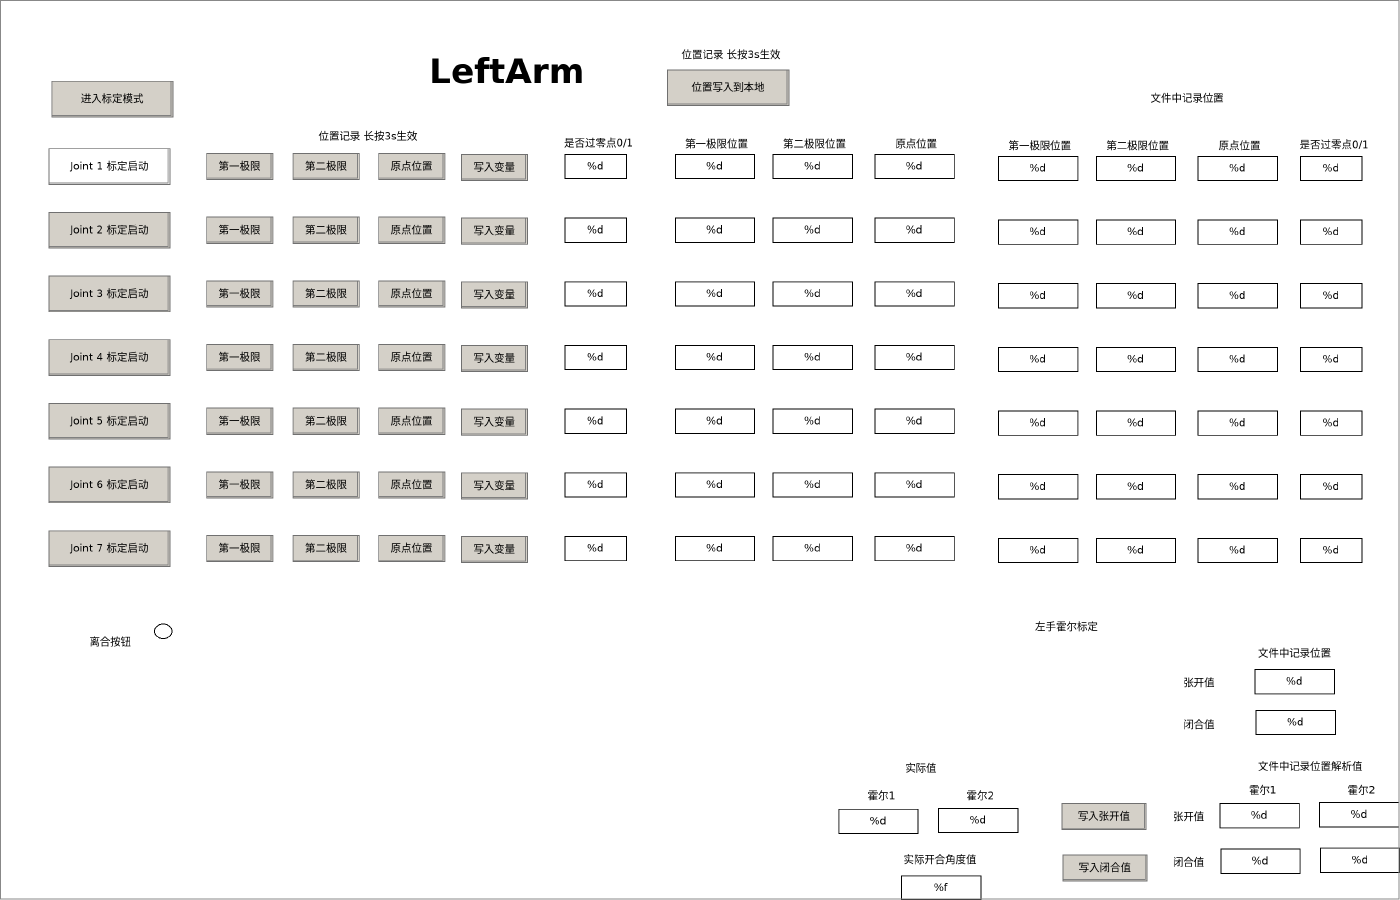
VISUALIZATION LeftArmCali  // 1473x947
    Button (54,85 128x38), "进入标定模式", colour toggle: GVL_armCali.g_armEnterCaliMode[1]
        toggle GVL_armCali.g_armEnterCaliMode[1]
    Button (51,156 128x38), "Joint 1 标定启动", colour toggle: GVL_armCali.g_jointIntoCaliState[1][1]
        toggle GVL_armCali.g_jointIntoCaliState[1][1]
    Label (435,49 197x52), "LeftArm"
    Button (51,223 128x38), "Joint 2 标定启动", colour toggle: GVL_armCali.g_jointIntoCaliState[1][2]
        toggle GVL_armCali.g_jointIntoCaliState[1][2]
    Button (217,161 70x28), "第一极限", colour toggle: GVL_armCali.g_linkEncFristCaliTrigger[1][1]
        tap GVL_armCali.g_linkEncFristPosCali[1][1]
    Button (308,161 70x28), "第二极限", colour toggle: GVL_armCali.g_linkEncSecondCaliTrigger[1][1]
        tap GVL_armCali.g_linkEncSecondPosCali[1][1]
    Rectangle (594,162 65x26), "%d", text variable: GVL_armCali.g_linkZeroCrossOrNot[1][1]
    Label (589,139 82x23), "是否过零点0/1"
    Rectangle (710,162 84x26), "%d", text variable: GVL_armCali.g_linkLimitFristPos[1][1]
    Label (713,140 82x23), "第一极限位置"
    Rectangle (813,162 84x26), "%d", text variable: GVL_armCali.g_linkLimitSecondPos[1][1]
    Label (816,140 82x23), "第二极限位置"
    Label (312,132 150x23), "位置记录 长按3s生效"
    Rectangle (920,162 84x26), "%d", text variable: GVL_armCali.g_linkHomePos[1][1]
    Label (923,140 82x23), "原点位置"
    Button (398,161 70x28), "原点位置", colour toggle: GVL_armCali.g_linkEncHomePosCaliTrigger[1][1]
        tap GVL_armCali.g_linkEncHomePosCali[1][1]
    Button (702,73 128x38), "位置写入到本地", colour toggle: GVL_armCali.g_caliDataWriteTrigger
        tap GVL_armCali.g_caliDataWrite
    Label (694,46 150x23), "位置记录 长按3s生效"
    Button (217,228 70x28), "第一极限", colour toggle: GVL_armCali.g_linkEncFristCaliTrigger[1][2]
        tap GVL_armCali.g_linkEncFristPosCali[1][2]
    Button (308,228 70x28), "第二极限", colour toggle: GVL_armCali.g_linkEncSecondCaliTrigger[1][2]
        tap GVL_armCali.g_linkEncSecondPosCali[1][2]
    Rectangle (594,229 65x26), "%d", text variable: GVL_armCali.g_linkZeroCrossOrNot[1][2]
    Rectangle (710,229 84x26), "%d", text variable: GVL_armCali.g_linkLimitFristPos[1][2]
    Rectangle (813,229 84x26), "%d", text variable: GVL_armCali.g_linkLimitSecondPos[1][2]
    Rectangle (920,229 84x26), "%d", text variable: GVL_armCali.g_linkHomePos[1][2]
    Button (398,228 70x28), "原点位置", colour toggle: GVL_armCali.g_linkEncHomePosCaliTrigger[1][2]
        tap GVL_armCali.g_linkEncHomePosCali[1][2]
    Button (51,290 128x38), "Joint 3 标定启动", colour toggle: GVL_armCali.g_jointIntoCaliState[1][3]
        toggle GVL_armCali.g_jointIntoCaliState[1][3]
    Button (217,295 70x28), "第一极限", colour toggle: GVL_armCali.g_linkEncFristCaliTrigger[1][3]
        tap GVL_armCali.g_linkEncFristPosCali[1][3]
    Button (308,295 70x28), "第二极限", colour toggle: GVL_armCali.g_linkEncSecondCaliTrigger[1][3]
        tap GVL_armCali.g_linkEncSecondPosCali[1][3]
    Rectangle (594,296 65x26), "%d", text variable: GVL_armCali.g_linkZeroCrossOrNot[1][3]
    Rectangle (710,296 84x26), "%d", text variable: GVL_armCali.g_linkLimitFristPos[1][3]
    Rectangle (813,296 84x26), "%d", text variable: GVL_armCali.g_linkLimitSecondPos[1][3]
    Rectangle (920,296 84x26), "%d", text variable: GVL_armCali.g_linkHomePos[1][3]
    Button (398,295 70x28), "原点位置", colour toggle: GVL_armCali.g_linkEncHomePosCaliTrigger[1][3]
        tap GVL_armCali.g_linkEncHomePosCali[1][3]
    Button (51,357 128x38), "Joint 4 标定启动", colour toggle: GVL_armCali.g_jointIntoCaliState[1][4]
        toggle GVL_armCali.g_jointIntoCaliState[1][4]
    Button (217,362 70x28), "第一极限", colour toggle: GVL_armCali.g_linkEncFristCaliTrigger[1][4]
        tap GVL_armCali.g_linkEncFristPosCali[1][4]
    Button (308,362 70x28), "第二极限", colour toggle: GVL_armCali.g_linkEncSecondCaliTrigger[1][4]
        tap GVL_armCali.g_linkEncSecondPosCali[1][4]
    Rectangle (594,363 65x26), "%d", text variable: GVL_armCali.g_linkZeroCrossOrNot[1][4]
    Rectangle (710,363 84x26), "%d", text variable: GVL_armCali.g_linkLimitFristPos[1][4]
    Rectangle (813,363 84x26), "%d", text variable: GVL_armCali.g_linkLimitSecondPos[1][4]
    Rectangle (920,363 84x26), "%d", text variable: GVL_armCali.g_linkHomePos[1][4]
    Button (398,362 70x28), "原点位置", colour toggle: GVL_armCali.g_linkEncHomePosCaliTrigger[1][4]
        tap GVL_armCali.g_linkEncHomePosCali[1][4]
    Button (51,424 128x38), "Joint 5 标定启动", colour toggle: GVL_armCali.g_jointIntoCaliState[1][5]
        toggle GVL_armCali.g_jointIntoCaliState[1][5]
    Button (217,429 70x28), "第一极限", colour toggle: GVL_armCali.g_linkEncFristCaliTrigger[1][5]
        tap GVL_armCali.g_linkEncFristPosCali[1][5]
    Button (308,429 70x28), "第二极限", colour toggle: GVL_armCali.g_linkEncSecondCaliTrigger[1][5]
        tap GVL_armCali.g_linkEncSecondPosCali[1][5]
    Rectangle (594,430 65x26), "%d", text variable: GVL_armCali.g_linkZeroCrossOrNot[1][5]
    Rectangle (710,430 84x26), "%d", text variable: GVL_armCali.g_linkLimitFristPos[1][5]
    Rectangle (813,430 84x26), "%d", text variable: GVL_armCali.g_linkLimitSecondPos[1][5]
    Rectangle (920,430 84x26), "%d", text variable: GVL_armCali.g_linkHomePos[1][5]
    Button (398,429 70x28), "原点位置", colour toggle: GVL_armCali.g_linkEncHomePosCaliTrigger[1][5]
        tap GVL_armCali.g_linkEncHomePosCali[1][5]
    Button (51,491 128x38), "Joint 6 标定启动", colour toggle: GVL_armCali.g_jointIntoCaliState[1][6]
        toggle GVL_armCali.g_jointIntoCaliState[1][6]
    Button (217,496 70x28), "第一极限", colour toggle: GVL_armCali.g_linkEncFristCaliTrigger[1][6]
        tap GVL_armCali.g_linkEncFristPosCali[1][6]
    Button (308,496 70x28), "第二极限", colour toggle: GVL_armCali.g_linkEncSecondCaliTrigger[1][6]
        tap GVL_armCali.g_linkEncSecondPosCali[1][6]
    Rectangle (594,497 65x26), "%d", text variable: GVL_armCali.g_linkZeroCrossOrNot[1][6]
    Rectangle (710,497 84x26), "%d", text variable: GVL_armCali.g_linkLimitFristPos[1][6]
    Rectangle (813,497 84x26), "%d", text variable: GVL_armCali.g_linkLimitSecondPos[1][6]
    Rectangle (920,497 84x26), "%d", text variable: GVL_armCali.g_linkHomePos[1][6]
    Button (398,496 70x28), "原点位置", colour toggle: GVL_armCali.g_linkEncHomePosCaliTrigger[1][6]
        tap GVL_armCali.g_linkEncHomePosCali[1][6]
    Button (51,558 128x38), "Joint 7 标定启动", colour toggle: GVL_armCali.g_jointIntoCaliState[1][7]
        toggle GVL_armCali.g_jointIntoCaliState[1][7]
    Button (217,563 70x28), "第一极限", colour toggle: GVL_armCali.g_linkEncFristCaliTrigger[1][7]
        tap GVL_armCali.g_linkEncFristPosCali[1][7]
    Button (308,563 70x28), "第二极限", colour toggle: GVL_armCali.g_linkEncSecondCaliTrigger[1][7]
        tap GVL_armCali.g_linkEncSecondPosCali[1][7]
    Rectangle (594,564 65x26), "%d", text variable: GVL_armCali.g_linkZeroCrossOrNot[1][7]
    Rectangle (710,564 84x26), "%d", text variable: GVL_armCali.g_linkLimitFristPos[1][7]
    Rectangle (813,564 84x26), "%d", text variable: GVL_armCali.g_linkLimitSecondPos[1][7]
    Rectangle (920,564 84x26), "%d", text variable: GVL_armCali.g_linkHomePos[1][7]
    Button (398,563 70x28), "原点位置", colour toggle: GVL_armCali.g_linkEncHomePosCaliTrigger[1][7]
        tap GVL_armCali.g_linkEncHomePosCali[1][7]
    Rectangle (1050,164 84x26), "%d", text variable: GVL_ArmJointCaliData.g_minLinkEncoder[1,1]
    Label (1053,142 82x23), "第一极限位置"
    Rectangle (1153,164 84x26), "%d", text variable: GVL_ArmJointCaliData.g_maxLinkEncoder[1,1]
    Label (1156,142 82x23), "第二极限位置"
    Rectangle (1260,164 84x26), "%d", text variable: GVL_ArmJointCaliData.g_caliLinkEncoder[1,1]
    Label (1263,142 82x23), "原点位置"
    Rectangle (1050,231 84x26), "%d", text variable: GVL_ArmJointCaliData.g_minLinkEncoder[1,2]
    Rectangle (1153,231 84x26), "%d", text variable: GVL_ArmJointCaliData.g_maxLinkEncoder[1,2]
    Rectangle (1260,231 84x26), "%d", text variable: GVL_ArmJointCaliData.g_caliLinkEncoder[1,2]
    Rectangle (1050,298 84x26), "%d", text variable: GVL_ArmJointCaliData.g_minLinkEncoder[1,3]
    Rectangle (1153,298 84x26), "%d", text variable: GVL_ArmJointCaliData.g_maxLinkEncoder[1,3]
    Rectangle (1260,298 84x26), "%d", text variable: GVL_ArmJointCaliData.g_caliLinkEncoder[1,3]
    Rectangle (1050,365 84x26), "%d", text variable: GVL_ArmJointCaliData.g_minLinkEncoder[1,4]
    Rectangle (1153,365 84x26), "%d", text variable: GVL_ArmJointCaliData.g_maxLinkEncoder[1,4]
    Rectangle (1260,365 84x26), "%d", text variable: GVL_ArmJointCaliData.g_caliLinkEncoder[1,4]
    Rectangle (1050,432 84x26), "%d", text variable: GVL_ArmJointCaliData.g_minLinkEncoder[1,5]
    Rectangle (1153,432 84x26), "%d", text variable: GVL_ArmJointCaliData.g_maxLinkEncoder[1,5]
    Rectangle (1260,432 84x26), "%d", text variable: GVL_ArmJointCaliData.g_caliLinkEncoder[1,5]
    Rectangle (1050,499 84x26), "%d", text variable: GVL_ArmJointCaliData.g_minLinkEncoder[1,6]
    Rectangle (1153,499 84x26), "%d", text variable: GVL_ArmJointCaliData.g_maxLinkEncoder[1,6]
    Rectangle (1260,499 84x26), "%d", text variable: GVL_ArmJointCaliData.g_caliLinkEncoder[1,6]
    Rectangle (1050,566 84x26), "%d", text variable: GVL_ArmJointCaliData.g_minLinkEncoder[1,7]
    Rectangle (1153,566 84x26), "%d", text variable: GVL_ArmJointCaliData.g_maxLinkEncoder[1,7]
    Rectangle (1260,566 84x26), "%d", text variable: GVL_ArmJointCaliData.g_caliLinkEncoder[1,7]
    Label (1174,92 150x23), "文件中记录位置"
    Rectangle (1368,164 65x26), "%d", text variable: GVL_ArmJointCaliData.g_linkEncZeroCross[1,1]
    Label (1363,141 82x23), "是否过零点0/1"
    Rectangle (1368,231 65x26), "%d", text variable: GVL_ArmJointCaliData.g_linkEncZeroCross[1,2]
    Rectangle (1368,298 65x26), "%d", text variable: GVL_ArmJointCaliData.g_linkEncZeroCross[1,3]
    Rectangle (1368,365 65x26), "%d", text variable: GVL_ArmJointCaliData.g_linkEncZeroCross[1,4]
    Rectangle (1368,432 65x26), "%d", text variable: GVL_ArmJointCaliData.g_linkEncZeroCross[1,5]
    Rectangle (1368,499 65x26), "%d", text variable: GVL_ArmJointCaliData.g_linkEncZeroCross[1,6]
    Rectangle (1368,566 65x26), "%d", text variable: GVL_ArmJointCaliData.g_linkEncZeroCross[1,7]
    Button (485,162 70x28), "写入变量", colour toggle: GVL_armCali.g_linkPosWriteCaliDataTrigger[1][1]
        tap GVL_armCali.g_linkPosWriteCaliData[1][1]
    Button (485,229 70x28), "写入变量", colour toggle: GVL_armCali.g_linkPosWriteCaliDataTrigger[1][2]
        tap GVL_armCali.g_linkPosWriteCaliData[1][2]
    Button (485,296 70x28), "写入变量", colour toggle: GVL_armCali.g_linkPosWriteCaliDataTrigger[1][3]
        tap GVL_armCali.g_linkPosWriteCaliData[1][3]
    Button (485,363 70x28), "写入变量", colour toggle: GVL_armCali.g_linkPosWriteCaliDataTrigger[1][4]
        tap GVL_armCali.g_linkPosWriteCaliData[1][4]
    Button (485,430 70x28), "写入变量", colour toggle: GVL_armCali.g_linkPosWriteCaliDataTrigger[1][5]
        tap GVL_armCali.g_linkPosWriteCaliData[1][5]
    Button (485,497 70x28), "写入变量", colour toggle: GVL_armCali.g_linkPosWriteCaliDataTrigger[1][6]
        tap GVL_armCali.g_linkPosWriteCaliData[1][6]
    Button (485,564 70x28), "写入变量", colour toggle: GVL_armCali.g_linkPosWriteCaliDataTrigger[1][7]
        tap GVL_armCali.g_linkPosWriteCaliData[1][7]
    Label (76,664 80x23), "离合按钮"
    Ellipse (162,656 19x16), colour toggle: GVL_IO.g_clutchSingle[1]
    Rectangle (1283,845 84x26), "%d", text variable: GVL_armCali.g_minArmHallCaliAnalysis[1][1]
    Rectangle (1388,844 84x26), "%d", text variable: GVL_armCali.g_minArmHallCaliAnalysis[1][2]
    Label (1082,648 80x23), "左手霍尔标定"
    Label (1308,676 108x23), "文件中记录位置"
    Label (1303,820 51x23), "霍尔1"
    Label (1407,820 51x23), "霍尔2"
    Rectangle (1284,893 84x26), "%d", text variable: GVL_armCali.g_maxArmHallCaliAnalysis[1][1]
    Rectangle (1389,892 84x26), "%d", text variable: GVL_armCali.g_maxArmHallCaliAnalysis[1][2]
    Label (1225,848 51x23), "张开值"
    Label (1225,896 51x23), "闭合值"
    Label (915,797 108x23), "实际值"
    Rectangle (882,851 84x26), "%d", text variable: MasterArmControl.m_masterRobot.m_masterArms[1].m_gripAngleCalc.m_gripHighHallSenorValue
    Rectangle (987,850 84x26), "%d", text variable: MasterArmControl.m_masterRobot.m_masterArms[1].m_gripAngleCalc.m_gripLowHallSenorValue
    Label (902,826 51x23), "霍尔1"
    Label (1006,826 51x23), "霍尔2"
    Rectangle (948,921 84x26), "%f", text variable: MasterArmControl.m_masterRobot.m_masterArms[1].m_gripAngle
    Label (935,893 108x23), "实际开合角度值"
    Button (1117,845 89x28), "写入张开值", colour toggle: GVL_armCali.g_masterArmHallCaliTrigger[1][1]
        tap GVL_armCali.g_masterArmHallCali[1][1]
    Button (1118,899 89x28), "写入闭合值", colour toggle: GVL_armCali.g_masterArmHallCaliTrigger[1][2]
        tap GVL_armCali.g_masterArmHallCali[1][2]
    Rectangle (1320,704 84x26), "%d", text variable: GVL_ArmJointCaliData.g_minHallSensorValue[1]
    Label (1236,707 51x23), "张开值"
    Label (1236,751 51x23), "闭合值"
    Rectangle (1321,747 84x26), "%d", text variable: GVL_ArmJointCaliData.g_maxHallSensorValue[1]
    Label (1314,795 129x23), "文件中记录位置解析值"
END_VISUALIZATION

(* stored: Version 1.1.0.1, ProductVersion 3.1.4024.11
   Visu LeftArmCali: Id {9cbc862b-ed55-45e4-b3ed-690df0b5758a} *)
